# EPICS substitutions: db/Beckhoff_9XXX/ecmcEL9110.substitutions
file "ecmcEL9110-chX.template"
{
  pattern {CH_ID}
          {01   }
}
